// TIA Portal V16 export
// export: Created 2021-08-10T09:05:00.3999489Z, ExportSetting WithDefaults, WithReadOnly, DisplayName Totally Integrated Automation Portal, DisplayVersion V16, DisplayName TIA Portal Version Control Interface, DisplayVersion V16, DisplayName TIA Portal Openness, DisplayVersion V16, DisplayName TIA Portal Teamcenter Gateway, DisplayVersion V16, DisplayName SINAMICS Startdrive Advanced, DisplayVersion V16, DisplayName SINAMICS Startdrive G130, G150, S120, S150, SINAMICS MV, S210, DisplayVersion V16, DisplayName SINAMICS Startdrive G110M, G120, G120C, G120D, G120P, DisplayVersion V16, DisplayName STEP 7 Professional, DisplayVersion V16, DisplayName STEP 7 Safety, DisplayVersion V16, DisplayName WinCC Unified SCADA Engineering System, DisplayVersion V16
FUNCTION "fcStepChooser" : Int   // FC185, SCL
{ S7_Optimized_Access := 'TRUE' }
VERSION : 0.0
// stored: AutoNumber false, CodeModifiedDate 2021-07-03T08:38:37.9433229Z, CompileDate 2021-07-03T08:38:37.9433229Z, CreationDate 2020-02-26T10:04:39.2339296Z, HandleErrorsWithinBlock false, InterfaceModifiedDate 2016-08-14T20:38:19.3457853Z, IsConsistent true, IsIECCheckEnabled false, IsKnowHowProtected false, IsWriteProtected false, LibraryConformanceStatus The object is library-conformant., LibraryType fcStepChooser V 3.0.1, LibraryTypeVersionGuid 8b64a3a6-6372-455a-bcc3-1a11207f1451, ModifiedDate 2021-07-03T08:38:37.9433229Z, ParameterModified 2016-08-14T20:38:19.3254825Z, PLCSimAdvancedSupport true, SetENOAutomatically true, StructureModified 2016-08-14T20:38:19.3457853Z, UDAEnableTagReadback false
   VAR_INPUT
      bCondition : Bool;
      iTrueStep : Int;
      iFalseStep : Int;
   END_VAR
   VAR_TEMP
      iResult : Int;
   END_VAR
BEGIN

       IF #bCondition THEN
           #iResult:=#iTrueStep;
       ELSE
           #iResult:=#iFalseStep;
       END_IF;
       ENO:=true;
       #fcStepChooser:=#iResult;
END_FUNCTION
